// TwinCAT 3 PLC project ABB_ACS380_Demo
// ProgramVersion: 3.1.4024.0
// libraries:
//   Tc2_Standard, * (Beckhoff Automation GmbH)
//   Tc2_System, * (Beckhoff Automation GmbH)
//   Tc3_Module, * (Beckhoff Automation GmbH)
// project tree:
//   DUTs/ ABB_ACS380.TcDUT, ABB_ControlWord.TcDUT, ABB_StatusWord.TcDUT
//   / PlcTask.TcTTO
//   POUs/ MAIN.TcPOU
// real-time tasks:
//   TASK Job Task: cycle default, priority 32
//   TASK PlcTask: cycle T#10ms, priority 20, ADS port 350
// I/O:
//   DEVICE Device 2 (EtherCAT), AmsNetId 10.0.2.193.3.1
//     Box 1 (FECA-01) [ABB FECA-01 EtherCAT adapter]
// variable links:
//   ABB ACS380 Demo/ABB ACS380 Demo Instance <-> Device 2 (EtherCAT)/Box 1 (FECA-01)
//     PlcTask Inputs/MAIN.ACS380.ComError <-> WcState/WcState
//     PlcTask Inputs/MAIN.ACS380.SpeedACT <-> TxPDO 6 map/vl velocity actual value
//     PlcTask Inputs/MAIN.ACS380.StatusWord <-> TxPDO 6 map/Statusword
//     PlcTask Outputs/MAIN.ACS380.ControlWord <-> RxPDO 6 map/Controlword
//     PlcTask Outputs/MAIN.ACS380.SpeedCMD <-> RxPDO 6 map/vl target velocity

CONFIGURATION ABB_ACS380_Demo
    RESOURCE PLC ON TwinCAT3
        TASK PlcTask(INTERVAL := T#10ms, PRIORITY := 20);
        PROGRAM MAIN WITH PlcTask : MAIN;
    END_RESOURCE
END_CONFIGURATION

// ---- DUTs/ABB_ACS380.TcDUT
TYPE ABB_ACS380 :
STRUCT
	StatusWord 	AT %I* 	: ABB_StatusWord;
	SpeedACT 	AT %I* 	: INT;
	ControlWord AT %Q* 	: ABB_ControlWord;
	SpeedCMD 	AT %Q* 	: INT; //P#50.04/50.07 = Frequency 0 to 60 = 0-60hz Reference P#46.02, = Speed -20000 to 20000 Reference Speed Scaling P#46.01
	ComError 	AT %I*	: BIT;
END_STRUCT
END_TYPE

// ---- DUTs/ABB_ControlWord.TcDUT
TYPE ABB_ControlWord :
STRUCT
	OFF1_CONTROL 		: BIT; //1=READY TO OPERATE, 0=STOP ALONG THE CURRENTLY ACTIVE DECEL RAMP
	OFF2_CONTROL 		: BIT; //1=CONTINUE OPERATION, 0=EMERGENCY OFF, COAST TO STOP
	OFF3_CONTROL 		: BIT; //1=CONTINUE OPERATION, 0=EMERGENCY STOP, STOP WITHIN THE TIME DEFINED BY THE DRIVE PARAMETER
	RUN 				: BIT; //1=OPERATION ENABLED, 0=OPERATION INHIBITED
	RAMP_OUT_ZERO 		: BIT; //1=NORMAL OPERATION RAMP FUNCTION GENERATOR, 0=FORCE RAMP FUNCTION OUTPUT TO 0
	RAMP_HOLD 			: BIT; //1=NORMAL OPERATION RAMP FUNCTION GENERATOR, 0=HALT RAMPING
	RAMP_IN_ZERO 		: BIT; //1=NORMAL OPERATION RAMP FUNCTION GENERATOR, 0=FORCE RAMP FUNCTION INPUT TO 0
	RESET 				: BIT; //0=>1 RESET ACTIVE FAULT
	INCHING_1 			: BIT; //1=ACCELERATE TO INCHING (JOGGING) SETPOINT 1, 0=DISABLED
	INCHING_2 			: BIT; //1=ACCELERATE TO INCHING (JOGGING) SETPOINT 2, 0=DISABLED
	REMOTE_CMD 			: BIT; //1=FIELDBUS CONTROL ENABLED, 0=LOCAL CONTROL
	EXT_CTRL_LOC 		: BIT; //NOT USED
	BIT_12 				: BIT; //NOT USED
	BIT_13 				: BIT; //NOT USED
	BIT_14 				: BIT; //NOT USED
	BIT_15 				: BIT; //NOT USED
END_STRUCT
END_TYPE

// ---- DUTs/ABB_StatusWord.TcDUT
TYPE ABB_StatusWord :
STRUCT
	RDY_ON 			: BIT; //1=READY TO SWITCH ON, 0=NOT READY
	RDY_RUN 		: BIT; //1=READY TO OPERATE, 0=OFF1 ACTIVE
	RDY_REF 		: BIT; //1=OPERATION ENABLED, 0=OPERATION INHIBITED
	TRIPPED 		: BIT; //1=FAULT, 0=NO FAULT
	OFF_2_STA 		: BIT; //1=OFF2 INACTIVE, 0=OFF2 ACTIVE
	OFF_3_STA 		: BIT; //1=OFF3 INACTIVE, 0=OFF3 ACTIVE
	SWC_ON_INHIB 	: BIT; //1=SWITCH-ON INHIBITED, 0=-
	WARNING 		: BIT; //1=ALARM/WARNING, 0=NO ALARM/WARNING
	AT_SETPOINT 	: BIT; //1=ACTUAL REFERENCE IS WITHIN TOLERANCE LIMITS
	REMOTE 			: BIT; //1=DRIVE CONTROL REMOTE, 0=DRIVE CONTROL LOCAL
	ABOVE_LIMIT 	: BIT; //1=FREQUENCY/SPEED EXCEEDS LIMITS 0=WITHIN LIMITS
	BIT_11 			: BIT; //1=EXTERNAL CONTROL EXT2 SELECTED, 0=EXTERNAL CONTROL EXT1 SELECTED
	BIT_12		 	: BIT; //1=EXTERNAL RUN ENABLE SIGNAL RECEIVED, 0=NO RUN ENABLE SIGNAL RECEIVED
	BIT_13 			: BIT; //NOT USED
	BIT_14 			: BIT; //NOT USED
	FBA_ERROR 		: BIT; //1=COMMUNICATION ERROR DETECTED, 0=COMMUNICATION OK	
END_STRUCT
END_TYPE

// ---- POUs/MAIN.TcPOU
PROGRAM MAIN
VAR
	
ACS380 		: ABB_ACS380;

xReady 		: BOOL;
xRun 		: BOOL;
xStop 		: BOOL;
xEstop		: BOOL;
xReset		: BOOL;
xJog		: BOOL;
xFaultPresent : BOOL;
iSpeedRef 	: INT;

END_VAR

//Need to be True
ACS380.ControlWord.REMOTE_CMD := TRUE;
ACS380.ControlWord.RAMP_OUT_ZERO := TRUE;
ACS380.ControlWord.RAMP_HOLD := TRUE;
ACS380.ControlWord.RAMP_IN_ZERO := TRUE;

//VFD Reset
	IF xReset THEN
		ACS380.ControlWord.RESET := TRUE;
	ELSE
		ACS380.ControlWord.RESET := FALSE;
	END_IF

//Stop Not Active
	IF NOT xStop AND NOT xEstop  THEN
		ACS380.ControlWord.OFF2_CONTROL := TRUE;
		ACS380.ControlWord.OFF3_CONTROL := TRUE;
	ELSE
		ACS380.ControlWord.OFF2_CONTROL := FALSE;
		ACS380.ControlWord.OFF3_CONTROL := FALSE;
	END_IF
	
//VFD Ready
	IF xReady AND ACS380.StatusWord.RDY_ON AND NOT ACS380.StatusWord.TRIPPED AND NOT xFaultPresent THEN
		ACS380.ControlWord.OFF1_CONTROL := TRUE;
	ELSE
		ACS380.ControlWord.OFF1_CONTROL := FALSE;
	END_IF
	
//Run VFD
	IF xRun AND ACS380.StatusWord.RDY_RUN THEN
		ACS380.ControlWord.RUN := TRUE;
	ELSE
		ACS380.ControlWord.RUN := FALSE;
	END_IF

//VFD Speed Command
	ACS380.SpeedCMD := iSpeedRef;
	
//VFD Fault
	IF ACS380.StatusWord.TRIPPED OR ACS380.ComError THEN
		xFaultPresent := TRUE;
	ELSIF xFaultPresent AND xReset THEN
		xFaultPresent := FALSE;
	END_IF

END_PROGRAM
